FUNCTION_BLOCK SOL_VIEWL (* Solenoid View with Local Data Publish/Subscribe *)
  (* Standard: 61499-1; Classification: View *)
  (* Version 0.0, 2004-09-23, JHC, Rockwell Automation, Adapted from MECH_VIEWL. *)
  (* Compiler header: package fb.rt.mva; import fb.rt.net.*; *)
  (* Compiler classdef: public class SOL_VIEWL extends FBMVCD *)
  (* Compiler Java Sun JDK 1.4.2 *)
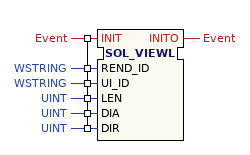
  EVENT_INPUT
    INIT WITH REND_ID, UI_ID, LEN, DIA, DIR; (* Initialize *)
  END_EVENT
  EVENT_OUTPUT
    INITO; (* Initialized *)
  END_EVENT
  VAR_INPUT
    REND_ID : WSTRING; (* Rendering Data Channel from Model *)
    UI_ID : WSTRING; (* User Input Channel to Model *)
    LEN : UINT; (* Length in Diameters *)
    DIA : UINT; (* Diameter *)
    DIR : UINT; (* Orientation:0=L/R,1=T/B,2=R/L,3=B/T *)
  END_VAR
  FBS
    REND : SUBL_1;
    VIEW : MECH_VIEW;
    UI : PUBL_1;
  END_FBS
  EVENT_CONNECTIONS
    INIT TO REND.INIT;
    REND.INITO TO VIEW.INIT;
    VIEW.INITO TO UI.INIT;
    UI.INITO TO INITO;
    REND.IND TO VIEW.REQ;
    VIEW.IND TO UI.REQ;
  END_CONNECTIONS
  DATA_CONNECTIONS
    REND.RD_1 TO VIEW.POS;
    VIEW.FAULT TO UI.SD_1;
    REND_ID TO REND.ID;
    UI_ID TO UI.ID;
    LEN TO VIEW.LEN;
    DIA TO VIEW.DIA;
    DIR TO VIEW.DIR;
    VSTYLE#SOLENOID TO VIEW.STYLE;
    COLOR#lightGray TO VIEW.WKPC;
    COLOR#darkGray TO VIEW.BKGD;
  END_CONNECTIONS
END_FUNCTION_BLOCK
